// TIA Portal V16 export
// export: Created 2023-03-29T11:03:27.427999Z, ExportSetting WithDefaults, DisplayName Totally Integrated Automation Portal, DisplayVersion V16 Update 6, DisplayName TIA Portal Version Control Interface, DisplayVersion V16 Update 2, DisplayName TIA Portal Openness, DisplayVersion V16 Update 6, DisplayName STEP 7 Professional, DisplayVersion V16 Update 6, DisplayName STEP 7 Safety, DisplayVersion V16, DisplayName WinCC Advanced, DisplayVersion V16 Update 6
DATA_BLOCK "dbModbusRTU_Reg"   // DB37
TITLE = Modbus RTU Data
{ S7_Optimized_Access := 'FALSE' }
AUTHOR : RTecmer
VERSION : 0.1
// Dane pomiarowe przekazane z bloku danych master modbus RTU
// stored: AutoNumber true, DBAccessibleFromOPCUA true, IsOnlyStoredInLoadMemory false, IsWriteProtectedInAS false
   VAR
      received_6_Wielkość_przeływu_Adres_0 { S7_SetPoint := 'True'} : "typeDataMPP04_Int";   // wielkość przepływu
      received_6_Licznik_objętość_VF_Adres_2 { S7_SetPoint := 'True'} : "typeDataMPP04_Int";   // licznik objętości VF
      received_6_Licznik_objętość_VR_Adres_4 { S7_SetPoint := 'True'} : "typeDataMPP04_Int";   // licznik objętości VR
      received_6_Licznik_różnicowy_VD_Adres_6 { S7_SetPoint := 'True'} : "typeDataMPP04_Int";   // licznik różnicy
      receive_6_Stan_licz_bjętości_GF_Adres_8 { S7_SetPoint := 'True'} : "typeDataMPP04_Int";   // licznik objetosci GF
      received_6_Stan_licz_bjętości_GR_Adres_10 { S7_SetPoint := 'True'} : "typeDataMPP04_Int";   // licznik objetości GR
      received_6_Stan_licz_rózicowego_obj_GD_Adres_12 { S7_SetPoint := 'True'} : "typeDataMPP04_Int";   // licznik róznicowy
      received_6_Stan_urządzenia_1000 { S7_SetPoint := 'True'} : "typeDataInverter_Word";   // stan urządzenia
      "Przepływomierz nr2" : Struct
         received_6_przeływu_VF_Adres_0 { S7_SetPoint := 'True'} : Real;
         received_6_objętość_VF_Adres_2 { S7_SetPoint := 'True'} : Real;
         "received_6_objętośc RF_Adres_4" { S7_SetPoint := 'True'} : Real;
         received_6_licznik_różnicowy_VD_Adres_7 { S7_SetPoint := 'True'} : Real;
         received_6_licznik_objętości_GF_Adres_8 { S7_SetPoint := 'True'} : Real;
         received_6_Licznik_objętości_GR_Adres_10 { S7_SetPoint := 'True'} : Real;
         received_6_Licznik_różnicowy_GD_Adres_12 { S7_SetPoint := 'True'} : Real;
         received_6_status_przepływomierza_Adres_1000 { S7_SetPoint := 'True'} : Word;
      END_STRUCT;
   END_VAR
BEGIN
END_DATA_BLOCK
